TYPE E_FillState :
(
    Idle   := 0,
    Dosing := 10,
    Done   := 20,
    Fault  := 99
) INT;
END_TYPE

(* stored: Version 1.1.0.1, ProductVersion 3.1.4024.0
   DUT E_FillState: Id {2e77a409-8c1b-4d53-9f26-b8410ce7d5a4} *)
